// TIA Portal V16 export
// export: Created 2021-07-12T14:47:21.2573633Z, ExportSetting WithDefaults, DisplayName Totally Integrated Automation Portal, DisplayVersion V16, DisplayName TIA Portal Version Control Interface, DisplayVersion V16, DisplayName TIA Portal Openness, DisplayVersion V16, DisplayName STEP 7 Professional, DisplayVersion V16, DisplayName STEP 7 Safety, DisplayVersion V16, DisplayName WinCC Professional, DisplayVersion V16
TYPE "SimaHydTO_typeHMIConnectionParameterSettingsCommands"
TITLE = SimaHydTO_typeHMIConnectionParameterSettingsCommands
// HMI interface: Parameter settings - Command (HMI -> PLC)
// stored: IsFailsafeCompliant false
   STRUCT
      Edit : Bool;
      Activate : Bool;
      Save : Bool;
      Restore : Bool;
      Abort : Bool;
      ApplyVChar : Bool;
      VCharSelector { S7_SetPoint := 'True'} : "SimaHydTO_typeHMIConnectionVCharSelectorCommand";
   END_STRUCT;
END_TYPE
